TYPE T_Ctrl_SIf_MER_In :
STRUCT
	/// Sensors for jam detection (option)
	a_bolJamSensor: ARRAY[1..cMAX_JAM_SENSORS] OF BASE_PLC.T_Ctrl_IoBool;
END_STRUCT
END_TYPE

(* stored: Version 1.1.0.1, ProductVersion 3.1.0.23
   DUT T_Ctrl_SIf_MER_In: Id {b86bd678-6cb9-46be-9f82-5c6e4f759512} *)
